{warning 'add method implementation '}
METHOD M_RunValve : BOOL
VAR_INPUT
	bStart	: BOOL;
END_VAR
VAR
	
END_VAR
M_RunValve := bStart;
END_METHOD

END_FUNCTION_BLOCK

// ---- RecipeControl/RecipeBlocks/Flush/FbFlush.TcPOU
FUNCTION_BLOCK FbFlush IMPLEMENTS IFlush
VAR_INPUT
END_VAR
VAR_OUTPUT
END_VAR
VAR
END_VAR

{warning 'add method implementation '}
METHOD Flush : BOOL
END_METHOD

{warning 'add property implementation'}
PROPERTY pEndFeedback : BOOL
GET
END_GET
END_PROPERTY

END_FUNCTION_BLOCK

// ---- RecipeControl/RecipeBlocks/Wait/fbWaitBlock.TcPOU
FUNCTION_BLOCK fbWaitBlock IMPLEMENTS IWaitBlock
VAR_INPUT
END_VAR
VAR_OUTPUT
END_VAR
VAR
END_VAR

END_FUNCTION_BLOCK
